PROGRAM P91_Monitoring
VAR
	TimeCycle			: TON;
	i 					: INT;
	idx					: INT;
	
	(*Utility Input*)
	bUtilityFault		: BYTE;	
END_VAR

//jhkang

(* Read from Utility Device*)
bUtilityFault		:= GVL_IO.aDigitalInputIO[7]; // 1~5 BYTE Operation, Normally Contacted

TimeCycle(IN:=TRUE, PT:=T#100MS); // 100MS Refresh Reading Time
IF TimeCycle.Q THEN
	TimeCycle(IN:=FALSE);
	
	// Reactor Ultimate Pressure Gauge
	GVL_IO.aMonitoring_PV[1] := GVL_IO.aAnalogInputIO[27] / GVL_CONSTANT.EL3064MaxValue * 10; //10Torr, 0~10V, Cal. x10
	// Exhaust Pressure Gauge
	GVL_IO.aMonitoring_PV[2] := GVL_IO.aAnalogInputIO[28] / GVL_CONSTANT.EL3064MaxValue * 1000; //1,000Torr, 0~10V, Cal. x1000
	
	GVL_IO.aAnalogOutputIO[27] := GVL_IO.aAnalogInputIO[28]; // Panel Meter Display
	
	// Double O-Ring(DOR) Gauge
	GVL_IO.aMonitoring_PV[3] := GVL_IO.aAnalogInputIO[29] / GVL_CONSTANT.EL3064MaxValueH * 100; //100kPa, 0~5V, Cal. x100
		
	//Gas Pressure 4 : N2, 5 : H2, 6 : NH3, 7 : SiH4
	GVL_IO.aMonitoring_PV[4] := GVL_IO.aAnalogInputIO[33] / GVL_CONSTANT.EL3064MaxValue * 6.89; // Cal. 6.89 bar
	GVL_IO.aMonitoring_PV[5] := GVL_IO.aAnalogInputIO[34] / GVL_CONSTANT.EL3064MaxValue * 6.89; // Cal. 6.89 bar
	GVL_IO.aMonitoring_PV[6] := GVL_IO.aAnalogInputIO[35] / GVL_CONSTANT.EL3064MaxValue * 6.89; // Cal. 6.89 bar
	GVL_IO.aMonitoring_PV[7] := GVL_IO.aAnalogInputIO[36] / GVL_CONSTANT.EL3064MaxValue * 6.89; // Cal. 6.89 bar
	
	// Cooling Water Temperature
	GVL_IO.aMonitoring_PV[8] := GVL_IO.aAnalogInputIO[37] * 0.1; // PT100, Shower Head, Cal. 0.1
	
END_IF

END_PROGRAM

(* stored: Version 1.1.0.1, ProductVersion 3.1.4024.15
   POU P91_Monitoring: Id {4f91223e-09c8-40bc-a729-040528b0179c}, SpecialFunc None *)
